INTERFACE I_Content EXTENDS I_ReadableData, I_WritableData

METHOD PUBLIC Accept
VAR_INPUT
	Visitor : I_ContentVisitor;
END_VAR
END_METHOD

PROPERTY PUBLIC Name : T_MAXSTRING
GET
END_GET
END_PROPERTY

END_INTERFACE

(* stored: Version 1.1.0.1, ProductVersion 3.1.4024.12
   Itf I_Content: Id {ac79f126-02b1-0527-0474-e319241b4fff}
   Method Accept: Id {956c3d1b-f47e-088a-2b6a-cda119d21818}
   Property Name: Id {52ea7131-31eb-095c-2b1b-24aafa810382}
   Get Get: Id {211a4fbf-0825-0d18-0755-a17e61f50184} *)
